Staubli VAL3: remErrConfig.pgx

program remErrConfig(string& sReturn[] (dimensions=1))
begin
  // Error raised when arm can't reach destination
  //
  logMsg("call remErrConfig")
  sReturn="ERROR 302"
  sReturn=sReturn+": Out of range or bad arm config."
  putln(sReturn)
  logMsg(sReturn)
end
